FUNCTION_BLOCK EL4112
VAR
	_io : EL4xx2_Data;
	{attribute addProperty Name "WcState"}
	_wcState : WcStateBase;
	{attribute addProperty Name "Info data"}
	_infoData : InfoDataAds;
END_VAR

PROPERTY IO : REFERENCE TO EL4xx2_Data
GET
IO REF= _io;
END_GET
END_PROPERTY

PROPERTY WcState : REFERENCE TO WcStateBase
GET
WcState REF= _wcState;
END_GET
END_PROPERTY

END_FUNCTION_BLOCK

(* stored: Version 1.1.0.1, ProductVersion 3.1.4024.9
   POU EL4112: Id {1b44dac8-113e-0369-3fd2-42201f2cf614}, SpecialFunc None
   Property IO: Id {1da3983a-121d-0476-2d91-33f1d1eb136e}
   Get Get: Id {cb61b6ba-2977-07cb-06cc-b3f55e8e9fbd}
   Property WcState: Id {74b8ac2b-c030-04c5-06f4-f146952db2e6}
   Get Get: Id {2e5bcbcf-1433-06d5-0759-270fe606c06b} *)
